PROGRAM P_ServoControl
VAR
	mc_powerSim1 :MC_power;
	mc_powerSim2 :MC_power;
	mc_MoveAbs1 :mc_moveAbsolute;
	mc_MoveAbs2 :mc_moveAbsolute;

	
	b_moveready: BOOL;
	TargetPos: LREAL;
END_VAR

IF io.PowerEnabled THEN
mc_powersim1(Axis:=io.Simdrive1, Enable := TRUE, Enable_positive := TRUE,Enable_negative := TRUE);
mc_powersim2(Axis:=io.Simdrive2, Enable := TRUE, Enable_positive := TRUE,Enable_negative := TRUE);
ELSE
	mc_powersim1(Axis:=io.Simdrive1, Enable := FALSE);
	mc_powersim2(Axis:=io.Simdrive2, Enable := FALSE);
	
END_IF

IF b_moveready THEN
	mc_moveAbs1(Axis := io.Simdrive1, Execute := TRUE, Position := TargetPos, Velocity := 1000,);
	b_moveready := FALSE;
ELSE
	mc_moveAbs1(Axis := io.Simdrive1, Execute := FALSE, Position := TargetPos, Velocity := 1000,);
END_IF

END_PROGRAM

(* stored: Version 1.1.0.1, ProductVersion 3.1.4024.3
   POU P_ServoControl: Id {140e10dd-763e-477f-a56d-97df28e55045}, SpecialFunc None *)
